// TIA Portal V17 export
// export: Created 2026-04-13T11:12:44.4988562Z, ExportSetting WithDefaults, DisplayName Totally Integrated Automation Portal, DisplayVersion V17 Update 4, DisplayName TIA Portal Openness, DisplayVersion V17 Update 4, DisplayName TIA Portal Version Control Interface, DisplayVersion V17, DisplayName SINAMICS Startdrive Advanced, DisplayVersion V17, DisplayName SINAMICS Startdrive G130, G150, S120, S150, SINAMICS MV, S210, DisplayVersion V17, DisplayName SINAMICS Startdrive G110M, G120, G120C, G120D, G120P, G115D, DisplayVersion V17, DisplayName STEP 7 Professional, DisplayVersion V17 Update 4, DisplayName STEP 7 Safety, DisplayVersion V17, DisplayName WinCC Professional, DisplayVersion V17 Update 4
DATA_BLOCK "C1-开式自动_DB"   // DB34
VERSION : 0.1
// stored: AutoNumber true, DBAccessibleFromOPCUA true, DBAccessibleFromWebserver true, InstanceOfName C1-开式自动, InstanceOfType FB
"C1-开式自动"
   // VAR
   //    开式自动喷雾 { S7_SetPoint := 'True'} : "开式自动喷雾块";
   //    KS开式自动自检 { S7_SetPoint := 'True'} : Bool;
   //    四参数辅助 { S7_SetPoint := 'True'} : "四参数辅助";
   //    TON1 { S7_SetPoint := 'True'} : TON_TIME;
   //    TON2 { S7_SetPoint := 'True'} : TON_TIME;
   //    TON3 { S7_SetPoint := 'True'} : TON_TIME;
   //    BD布袋反吹记录 { S7_SetPoint := 'True'} : "D3-布袋记录";
   // END_VAR
BEGIN
END_DATA_BLOCK
